FUNCTION_BLOCK FINAL FB_MiscInput EXTENDS FB_EventLogger                                            	
VAR_IN_OUT                                          	
	Control					: ST_System;            	//Machine Control Instance
END_VAR                                             	                                           	
VAR           
	_Input		AT %I*		: BOOL;						//Raw Input 1
	_Input2		AT %I*		: BOOL;						//Raw Input 2                                   	
	_ManOn					: BOOL;	     				//Manual On
	_ManOff					: BOOL;	     				//Manual Off
	_ForceOn				: BOOL;	     				//Force On
	_ForceOff				: BOOL;	     				//Force Off
	_Fault					: BOOL;	     				//Device Fault
	_SimInput				: BOOL;						//Simulates Input
	_FallingEdge			: BOOL;						//Falling Edge of Value Signal
	_RisingEdge				: BOOL;						//Raising Edge of Value Signal
	_DebounceOn_ET			: REAL;						//Debounce On Elapsed Time
	_DebounceOff_ET			: REAL;						//Debounce Off Elapsed Time
	_FaultTimer_ET			: REAL;						//Fault timer elapsed
	_EvaluationError		: BOOL;						//Evaluation Error
	_TestPulseGeneralFault	: BOOL;						//Test Pulse General Fault
	_TestPulse1Fault		: BOOL;						//Test Pulse 1 Fault
	_TestPulse2Fault		: BOOL;						//Test Pulse 2 Fault
	_Alarm					: BOOL;						//Device Alarm
	_Warning				: BOOL;						//Device Warning
	_AlarmNum				: DINT;						//Device Alarm Number
	_WarningNum				: DINT;						//Device Warning Number
	_ConfInput				: BOOL;						//Confirgured Input
	_DebounceOn_DN			: BOOL;						//Debounce On Timer is Done
	_DebounceOff_DN			: BOOL;						//Debounce Off Timer is Done
	_RiseEdge				: R_TRIG;					//Rising Edge Value Trigger
	_FallEdge				: F_TRIG;					//Falling Edge Value Trigger
	_Value		AT %Q*		: BOOL;						//Value of Input
	_R_Trig					: ARRAY[0..9] OF R_TRIG;	//Private Rising Edge Triggers
END_VAR
VAR PERSISTENT
	_Name					: STRING[15];				//Name for HMI
	_Description			: STRING[40];				//Description for HMI
	_AlarmMute				: BOOL;						//Alarm Mute
	_TypeConfig				: E_InputTypeConfig;		//Type congifuration
	_DebounceOn_PT			: REAL;						//Debounce on timer preset time
	_DebounceOff_PT			: REAL;						//Debounce off timer preset time
	_FaultTimer_PT			: REAL;						//Fault timer preset time
END_VAR

M_TypeConfig();
M_AlarmMonitor();
M_WarningMonitor();
M_UnlatchManuals();

//Debounce On Timer
IF _ConfInput = TRUE AND NOT _ForceOff AND NOT _ManOff THEN
	_DebounceOn_ET := _DebounceOn_ET + Control.SystemTime.ScanTime;
	_debounceOn_DN := _DebounceOn_ET > _DebounceOn_PT;
ELSE
	_debounceOn_DN := FALSE;
END_IF
IF _debounceOn_DN OR _ForceOn OR _ManOn THEN
	_Value := TRUE;
	_DebounceOff_ET := 0;
END_IF

//Debounce Off Timer
IF _ConfInput = FALSE AND NOT _ForceOn AND NOT _ManOn THEN
	_DebounceOff_ET := _DebounceOff_ET + Control.SystemTime.ScanTime;
	_debounceOff_DN := _DebounceOff_ET > _DebounceOff_PT;
ELSE
	_debounceOff_DN := FALSE;
END_IF
IF _debounceOff_DN OR _ForceOff OR _ManOff THEN
	_Value := FALSE;
	_DebounceOn_ET := 0;
END_IF

//Rising Edge Trigger 
_riseEdge(CLK := _Value);
_RisingEdge := _riseEdge.Q;

//Falling Edge Trigger
_fallEdge(CLK := _Value);
_FallingEdge := _fallEdge.Q;

{attribute 'monitoring' := 'variable'}
PROPERTY PUBLIC Alarm : Bool
GET
Alarm := _Alarm;
END_GET
END_PROPERTY

{attribute 'monitoring' := 'variable'}
PROPERTY PUBLIC AlarmMute : BOOL
SET
AlarmMute := _AlarmMute;
END_SET
END_PROPERTY

{attribute 'monitoring' := 'variable'}
PROPERTY PUBLIC AutoStandbyReset : Bool
GET
AutoStandbyReset := _ForceOff;
END_GET
SET
_ForceOff := AutoStandbyReset;
END_SET
END_PROPERTY

{attribute 'monitoring' := 'variable'}
PROPERTY PUBLIC DebounceOff_ET : real
GET
DebounceOff_ET := _DebounceOff_ET;
END_GET
END_PROPERTY

{attribute 'monitoring' := 'variable'}
PROPERTY PUBLIC DebounceOff_PT : real
GET
DebounceOff_PT := _DebounceOff_PT;
END_GET
SET
_DebounceOff_PT := DebounceOff_PT;
END_SET
END_PROPERTY

{attribute 'monitoring' := 'variable'}
PROPERTY PUBLIC DebounceOn_ET : real
GET
DebounceOn_ET := _DebounceOn_ET;
END_GET
END_PROPERTY

{attribute 'monitoring' := 'variable'}
PROPERTY PUBLIC DebounceOn_PT : real
GET
DebounceOn_PT := _DebounceOn_PT;
END_GET
SET
_DebounceOn_PT := DebounceOn_PT;
END_SET
END_PROPERTY

{attribute 'monitoring' := 'variable'}
PROPERTY PUBLIC Description : String[40]
GET
Description := _Description;
END_GET
SET
_Description := Description;
END_SET
END_PROPERTY

{attribute 'monitoring' := 'variable'}
PROPERTY PUBLIC EvaluationError : Bool
GET // PUBLIC
EvaluationError := _EvaluationError;
END_GET
SET
_EvaluationError := EvaluationError;
END_SET
END_PROPERTY

{attribute 'monitoring' := 'variable'}
PROPERTY PUBLIC FallingEdge : Bool
GET
FallingEdge := _FallingEdge;
END_GET
END_PROPERTY

{attribute 'monitoring' := 'variable'}
PROPERTY PUBLIC Fault : Bool
SET
_Fault := Fault;
END_SET
END_PROPERTY

{attribute 'monitoring' := 'variable'}
PROPERTY PUBLIC FaultTimer_ET : real
GET
FaultTimer_ET := _FaultTimer_ET;
END_GET
END_PROPERTY

{attribute 'monitoring' := 'variable'}
PROPERTY PUBLIC FaultTimer_PT : real
GET
FaultTimer_PT := _FaultTimer_PT;
END_GET
SET
_FaultTimer_PT := FaultTimer_PT;
END_SET
END_PROPERTY

{attribute 'monitoring' := 'variable'}
PROPERTY PUBLIC ForceOn : Bool
GET
ForceOn := _ForceOn;
END_GET
SET
_ForceOn := ForceOn;
END_SET
END_PROPERTY

{attribute 'monitoring' := 'variable'}
PROPERTY PUBLIC Input : Bool
GET
Input := _Input;
END_GET
SET // PUBLIC
_Input := Input;
END_SET
END_PROPERTY

{attribute 'monitoring' := 'variable'}
PROPERTY PUBLIC Input2 : Bool
GET
Input2 := _Input2;
END_GET
END_PROPERTY

METHOD PRIVATE M_AlarmMonitor
VAR_INPUT
END_VAR
VAR_INST
	_EvaluationError_TON		: 		TON;
END_VAR
VAR_INST // added by the converter: edge detectors and wires of the graphical bodies
    _w1, _w2, _w3, _w4, _w5 : BOOL;
    _rt1 : R_TRIG;
END_VAR
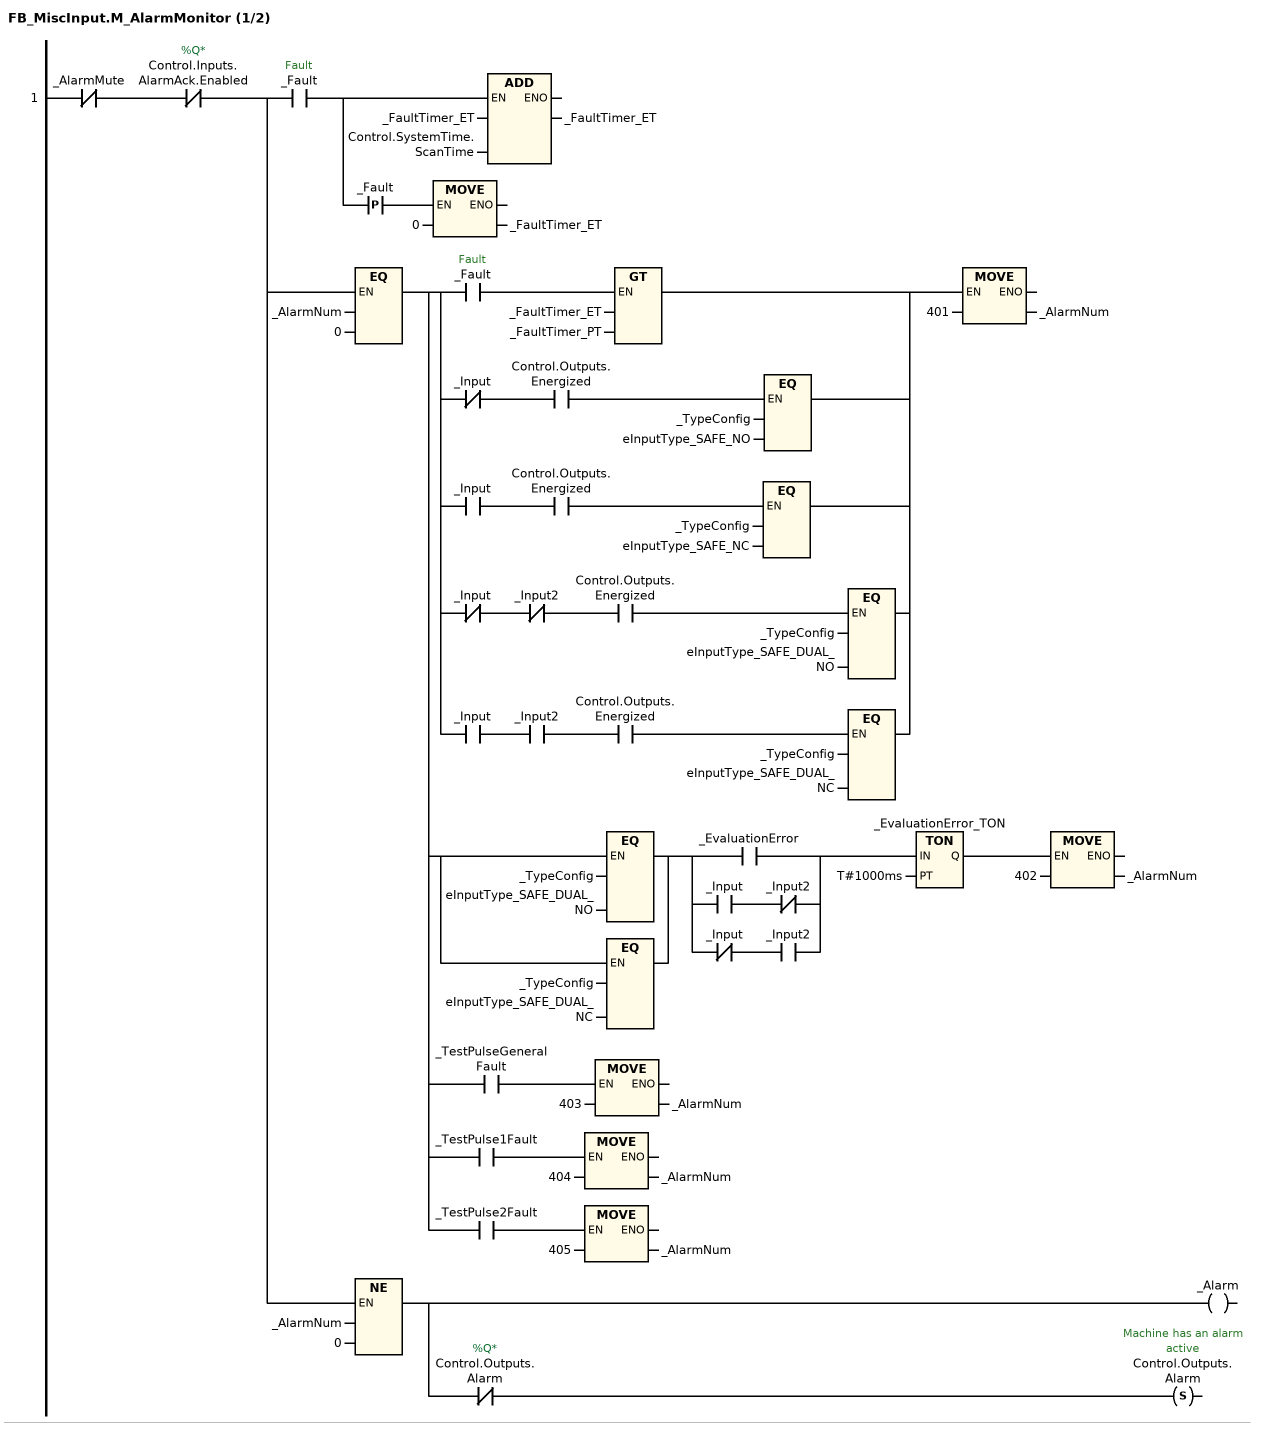
// NETWORK 1
//   Control.Inputs.AlarmAck.Enabled: AT %Q*
//   _Fault: Fault
//   _FaultTimer_ET: Fault timer elapsed
//   Control.SystemTime.ScanTime: Last scan time (Seconds)
//   _FaultTimer_PT: Fault timer preset time
//   Control.Outputs.Alarm: AT %Q* | Machine has an alarm active
_w1 := NOT _AlarmMute AND NOT Control.Inputs.AlarmAck.Enabled;
_w2 := _w1 AND _Fault;
IF _w2 THEN _FaultTimer_ET := _FaultTimer_ET + Control.SystemTime.ScanTime; END_IF
_rt1(CLK := _Fault);
IF _w2 AND _rt1.Q THEN _FaultTimer_ET := 0; END_IF
_w3 := _w1 AND _AlarmNum = 0;
IF _w3 AND _Fault AND _FaultTimer_ET > _FaultTimer_PT OR (_w3 AND NOT _Input) AND Control.Outputs.Energized AND _TypeConfig = eInputType_SAFE_NO OR (_w3 AND _Input) AND Control.Outputs.Energized AND _TypeConfig = eInputType_SAFE_NC OR (_w3 AND NOT _Input) AND NOT _Input2 AND Control.Outputs.Energized AND _TypeConfig = eInputType_SAFE_DUAL_NO OR (_w3 AND _Input) AND _Input2 AND Control.Outputs.Energized AND _TypeConfig = eInputType_SAFE_DUAL_NC THEN
    _AlarmNum := 401;
END_IF
_EvaluationError_TON(IN := (_w3 AND _TypeConfig = eInputType_SAFE_DUAL_NO OR _w3 AND _TypeConfig = eInputType_SAFE_DUAL_NC) AND (_EvaluationError OR _Input AND NOT _Input2 OR NOT _Input AND _Input2), PT := T#1000ms); // TON
IF _EvaluationError_TON.Q THEN _AlarmNum := 402; END_IF
IF _w3 AND _TestPulseGeneralFault THEN _AlarmNum := 403; END_IF
IF _w3 AND _TestPulse1Fault THEN _AlarmNum := 404; END_IF
IF _w3 AND _TestPulse2Fault THEN _AlarmNum := 405; END_IF
_w4 := _w1 AND _AlarmNum <> 0;
_Alarm := _w4;
Control.Outputs.Alarm S= _w4 AND NOT Control.Outputs.Alarm;

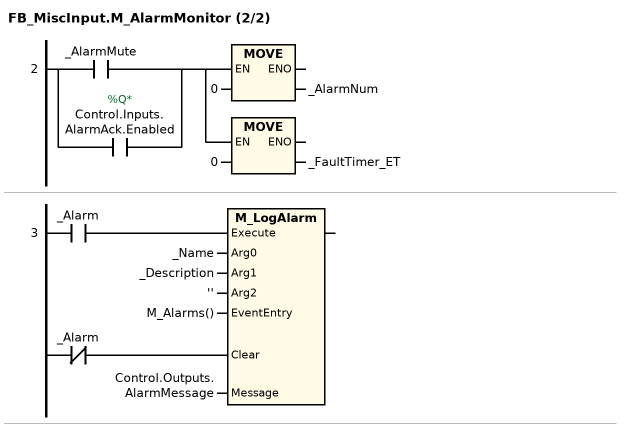
// NETWORK 2
//   Control.Inputs.AlarmAck.Enabled: AT %Q*
//   _FaultTimer_ET: Fault timer elapsed
_w5 := _AlarmMute OR Control.Inputs.AlarmAck.Enabled;
IF _w5 THEN _AlarmNum := 0; END_IF
IF _w5 THEN _FaultTimer_ET := 0; END_IF

// NETWORK 3
M_LogAlarm(Execute := _Alarm, Arg0 := _Name, Arg1 := _Description, Arg2 := '', EventEntry := M_Alarms(), Clear := NOT _Alarm, Message := Control.Outputs.AlarmMessage);
END_METHOD

METHOD PRIVATE M_Alarms : TcEventEntry
VAR_INPUT
END_VAR
CASE _AlarmNum OF
	401: M_Alarms:= TC_Events.TcMiscInput.A_401;//Alarm
	402: M_Alarms:= TC_Events.TcMiscInput.A_402;//Evaluation Error. Contact 1 or 2 failed to switch or switched too late			
	403: M_Alarms:= TC_Events.TcMiscInput.A_403;//Error in the test pulse wiring.
	404: M_Alarms:= TC_Events.TcMiscInput.A_404;//Channel 1 Input Test Pulse Error	
	405: M_Alarms:= TC_Events.TcMiscInput.A_405;//Channel 2 Input Test Pulse Error			
	406: M_Alarms:= TC_Events.TcMiscInput.A_406;//Expected to be ON Fault		
	407: M_Alarms:= TC_Events.TcMiscInput.A_407;//Expected to be OFF Fault						
ELSE
	M_Alarms:= TC_Events.TcMiscInput.A_Undefined;
END_CASE
END_METHOD

METHOD PRIVATE M_TypeConfig
VAR_INPUT
END_VAR
VAR_INST
END_VAR
CASE _TypeConfig OF
	eInputType_PLC_NO, eInputType_SAFE_NO : 
		IF _Input OR _SimInput THEN
			_ConfInput := TRUE;
		ELSE
			_ConfInput := FALSE;
		END_IF
	eInputType_PLC_NC, eInputType_SAFE_NC : 
		IF NOT _Input OR _SimInput THEN
			_ConfInput := TRUE;
		ELSE
			_ConfInput := FALSE;
		END_IF
	eInputType_SAFE_DUAL_NO : 
		IF _Input AND _Input2 THEN
			_ConfInput := TRUE;
		ELSE
			_ConfInput := FALSE;
		END_IF
	eInputType_SAFE_DUAL_NC : 
		IF NOT _Input AND NOT _Input2 THEN
			_ConfInput := TRUE;
		ELSE
			_ConfInput := FALSE;
		END_IF
	eInputType_SAFE_DUAL_NO_NC : 
		IF _Input AND NOT _Input2 THEN
			_ConfInput := TRUE;
		ELSE
			_ConfInput := FALSE;
		END_IF
END_CASE
END_METHOD

METHOD PRIVATE M_UnlatchManuals
VAR_INPUT
END_VAR
VAR_INST
END_VAR
VAR_INST // added by the converter: edge detectors and wires of the graphical bodies
    _rt1, _rt2, _rt3 : R_TRIG;
END_VAR
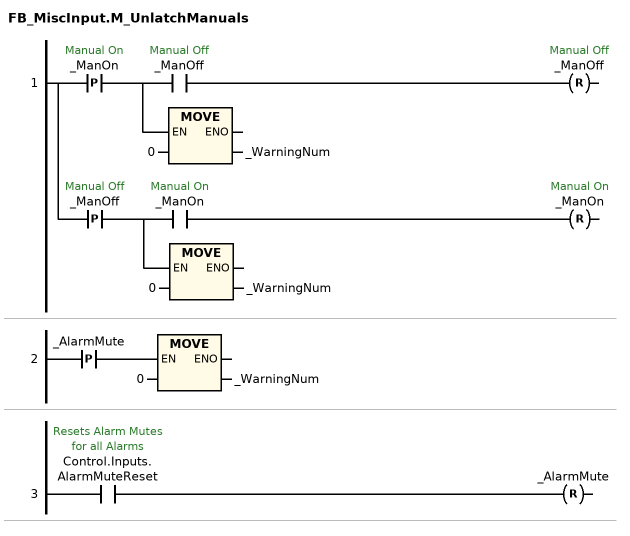
// NETWORK 1
//   _ManOn: Manual On
//   _ManOff: Manual Off
_rt1(CLK := _ManOn);
_ManOff R= _rt1.Q AND _ManOff;
IF _rt1.Q THEN _WarningNum := 0; END_IF
_rt2(CLK := _ManOff);
_ManOn R= _rt2.Q AND _ManOn;
IF _rt2.Q THEN _WarningNum := 0; END_IF

// NETWORK 2
_rt3(CLK := _AlarmMute);
IF _rt3.Q THEN _WarningNum := 0; END_IF

// NETWORK 3
//   Control.Inputs.AlarmMuteReset: Resets Alarm Mutes for all Alarms
_AlarmMute R= Control.Inputs.AlarmMuteReset;
END_METHOD

METHOD PRIVATE M_WarningMonitor
VAR_INPUT
END_VAR
VAR_INST
END_VAR
VAR_INST // added by the converter: edge detectors and wires of the graphical bodies
    _w1 : BOOL;
END_VAR
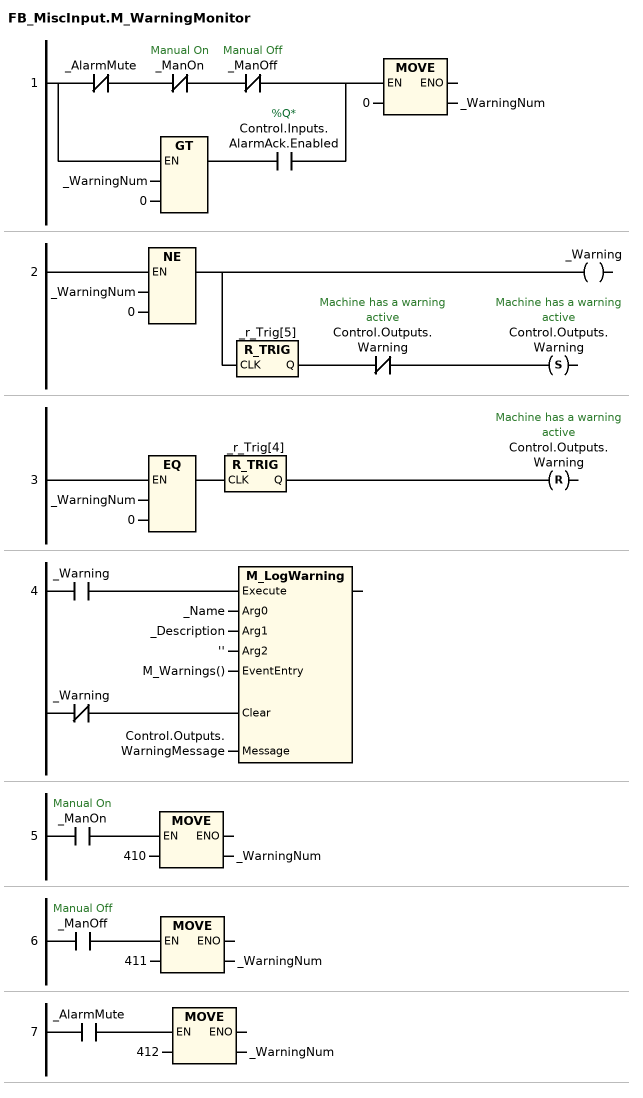
// NETWORK 1
//   _ManOn: Manual On
//   _ManOff: Manual Off
//   Control.Inputs.AlarmAck.Enabled: AT %Q*
IF NOT _AlarmMute AND NOT _ManOn AND NOT _ManOff OR _WarningNum > 0 AND Control.Inputs.AlarmAck.Enabled THEN
    _WarningNum := 0;
END_IF

// NETWORK 2
//   Control.Outputs.Warning: Machine has a warning active
_w1 := _WarningNum <> 0;
_Warning := _w1;
_r_Trig[5](CLK := _w1); // R_TRIG
Control.Outputs.Warning S= _r_Trig[5].Q AND NOT Control.Outputs.Warning;

// NETWORK 3
//   Control.Outputs.Warning: Machine has a warning active
_r_Trig[4](CLK := _WarningNum = 0); // R_TRIG
Control.Outputs.Warning R= _r_Trig[4].Q;

// NETWORK 4
M_LogWarning(Execute := _Warning, Arg0 := _Name, Arg1 := _Description, Arg2 := '', EventEntry := M_Warnings(), Clear := NOT _Warning, Message := Control.Outputs.WarningMessage);

// NETWORK 5
//   _ManOn: Manual On
IF _ManOn THEN _WarningNum := 410; END_IF

// NETWORK 6
//   _ManOff: Manual Off
IF _ManOff THEN _WarningNum := 411; END_IF

// NETWORK 7
IF _AlarmMute THEN _WarningNum := 412; END_IF
END_METHOD

METHOD PRIVATE M_Warnings : TcEventEntry
VAR_INPUT
END_VAR
CASE _WarningNum OF
	410: M_Warnings:= TC_Events.TcMiscInput.W_410;//Manual ON Enabled	
	411: M_Warnings:= TC_Events.TcMiscInput.W_411;//Manual OFF Enabled			
	412: M_Warnings:= TC_Events.TcMiscInput.W_412;//Alarm Mute Active						
ELSE
	M_Warnings:=  TC_Events.TcMiscInput.W_Undefined;
END_CASE
END_METHOD

{attribute 'monitoring' := 'variable'}
PROPERTY PUBLIC ManOff : Bool
GET
ManOff := _ManOff;
END_GET
SET
_ManOff := ManOff;
END_SET
END_PROPERTY

{attribute 'monitoring' := 'variable'}
PROPERTY PUBLIC ManOn : Bool
GET
ManOn := _ManOn;
END_GET
SET
_ManOn := ManOn;
END_SET
END_PROPERTY

{attribute 'monitoring' := 'variable'}
PROPERTY PUBLIC Name : String[15]
GET
Name := _Name;
END_GET
SET
_Name := Name;
END_SET
END_PROPERTY

{attribute 'monitoring' := 'variable'}
PROPERTY PUBLIC RisingEdge : Bool
GET
RisingEdge := _RisingEdge;
END_GET
END_PROPERTY

{attribute 'monitoring' := 'variable'}
PROPERTY PUBLIC SimInput : Bool
SET
_SimInput := SimInput;
END_SET
END_PROPERTY

{attribute 'monitoring' := 'variable'}
PROPERTY PUBLIC TestPulse1Fault : Bool
GET
TestPulse1Fault := _TestPulse1Fault;
END_GET
SET
_TestPulse1Fault := TestPulse1Fault;
END_SET
END_PROPERTY

{attribute 'monitoring' := 'variable'}
PROPERTY PUBLIC TestPulse2Fault : Bool
GET
TestPulse2Fault := _TestPulse2Fault;
END_GET
SET
_TestPulse2Fault := TestPulse2Fault;
END_SET
END_PROPERTY

{attribute 'monitoring' := 'variable'}
PROPERTY PUBLIC TestPulseGeneralFault : Bool
GET
TestPulseGeneralFault := _TestPulseGeneralFault;
END_GET
SET
_TestPulseGeneralFault := TestPulseGeneralFault;
END_SET
END_PROPERTY

{attribute 'monitoring' := 'variable'}
PROPERTY PUBLIC Value : Bool
GET
Value := _Value;
END_GET
SET
_Value := Value;
END_SET
END_PROPERTY

{attribute 'monitoring' := 'variable'}
PROPERTY PUBLIC Warning : Bool
GET
Warning := _Warning;
END_GET
END_PROPERTY

END_FUNCTION_BLOCK

(* stored: Version 1.1.0.1, ProductVersion 3.1.4024.3
   POU FB_MiscInput: Id {c0d88bc5-b182-49df-b578-ed0f16238807}, SpecialFunc None
   Property Alarm: Id {3658f6dc-6e01-4ab1-aa7a-12bbd299ad4b}
   Get Get: Id {6c509c0c-7480-4274-ae68-68e3a9df5369}
   Property AlarmMute: Id {ffa553a3-2559-4579-a69b-9f764a8d08ab}
   Set Set: Id {cf89d9e7-8292-4528-a66f-29cd89792830}
   Property AutoStandbyReset: Id {18cb0727-a662-4c09-8dbc-84357f54838e}
   Get Get: Id {b0a025ea-2b9e-400d-8a61-1d76b1ed73bf}
   Set Set: Id {b2ad94f4-5c45-4b2e-82a5-1581ac1c5dc8}
   Property DebounceOff_ET: Id {74509f44-dd39-4467-8d20-707144248c24}
   Get Get: Id {54d68720-48e0-4727-905c-29fbd4979d9a}
   Property DebounceOff_PT: Id {59f53b24-f1c7-4249-805f-05c62da47c84}
   Get Get: Id {8891ec69-8d1f-4c4a-b114-deeb08ce2fb7}
   Set Set: Id {ed01c235-50fd-48e7-b591-2a2a9a9e33ce}
   Property DebounceOn_ET: Id {41af56ee-a2d6-477e-b0cf-98933ddbaa42}
   Get Get: Id {cbd68782-1d64-467e-aabe-68254bed39b3}
   Property DebounceOn_PT: Id {251423d0-2084-4b2d-afa5-afd07bfcc653}
   Get Get: Id {a8f1dbac-0971-46e9-9af2-c1757fd9c4f5}
   Set Set: Id {d501fff4-40d2-4cda-bdf5-80cb053ebb49}
   Property Description: Id {0a20c4d0-0852-4169-8173-d3c2bd3caa54}
   Get Get: Id {124a4c05-8915-484c-b001-008a20669f39}
   Set Set: Id {f84e5111-a402-48fd-a46f-f4a9cee7eb8c}
   Property EvaluationError: Id {f8c56a30-f5c7-41f6-aee7-0206f6f8cd4e}
   Get Get: Id {38e8d71a-2fe3-43ac-aea2-c10b7579b2e9}
   Set Set: Id {ff11a864-f0e3-4f8f-acd7-475b40d97727}
   Property FallingEdge: Id {1dd8b317-91a8-4de8-b759-d4e8f3ca831a}
   Get Get: Id {e6170223-0c69-4d8c-8877-6cf3fd201983}
   Property Fault: Id {125dc8d1-6763-4ef4-93a0-c88b685b439a}
   Set Set: Id {ae2cc827-cc43-4139-bb37-9ded44db5652}
   Property FaultTimer_ET: Id {0fba5d22-2aeb-4884-b5c9-eb62bc396633}
   Get Get: Id {1111c4e2-66c0-4d9f-9925-39545e35947a}
   Property FaultTimer_PT: Id {d2d56292-bc61-416b-8e16-e19ad9993c6e}
   Get Get: Id {34faa55f-4d25-41b6-883c-99de9ba5fb41}
   Set Set: Id {daca9458-4a85-4640-982b-cf6448678cba}
   Property ForceOn: Id {0377b997-3862-47a0-95f4-b96c26817522}
   Get Get: Id {06c3b5dc-e414-4a3a-a58e-0c0a4672b0ad}
   Set Set: Id {a0ce7201-4ff4-408a-a056-42104c48bc78}
   Property Input: Id {488231ea-c389-4dd6-8b10-b85cda51d1dc}
   Get Get: Id {55032826-2e2a-4ab2-919c-0cd7931ef0fa}
   Set Set: Id {00a98704-90c3-4ab5-9755-e1394caca87d}
   Property Input2: Id {a441fdbc-27f5-4bd6-a1bf-204e52cb7712}
   Get Get: Id {a0d87452-58a1-4b2b-8b9c-f140e2cdba22}
   Method M_AlarmMonitor: Id {7ca0b0a4-1432-430e-b009-7d687ad3806f}
   Method M_Alarms: Id {c867b0f2-aa9f-49f4-96fa-dbbc2082d479}
   Method M_TypeConfig: Id {4a7e9782-dd7a-4141-992d-c79556985019}
   Method M_UnlatchManuals: Id {2bd763b3-55d1-4150-b0ec-e296a1f80358}
   Method M_WarningMonitor: Id {583cee2f-f972-4331-a8ee-8fba29d76a89}
   Method M_Warnings: Id {f0c100d2-055b-4c71-a5ca-5744cfb67d26}
   Property ManOff: Id {18c427a3-b5f4-49d8-8024-d24d3e51a681}
   Get Get: Id {2c36e6a8-0f41-487f-b4d1-51c40bc21ef1}
   Set Set: Id {2573b357-9d4f-41f5-8737-2fbb1dd13605}
   Property ManOn: Id {0e133ec4-1599-4ebb-b406-35e05fb2c0bb}
   Get Get: Id {7df83b3c-429d-496b-a33a-656de7942966}
   Set Set: Id {eba54b43-038e-46b3-bde0-df3e437c05f8}
   Property Name: Id {23ff72d4-11f9-447d-b9b1-0b8adf36daaa}
   Get Get: Id {17028a0b-910a-49b3-a4c1-72fd230b2f75}
   Set Set: Id {84d80d55-f619-4c80-ac5a-5c0f5305badd}
   Property RisingEdge: Id {97e0f4e1-a76f-4f1e-a85d-3e5217da4311}
   Get Get: Id {a415b987-98ac-4008-94ee-3e79e7da5f22}
   Property SimInput: Id {9ebabc78-61d5-4206-8c01-1ed75c8ddc37}
   Set Set: Id {79f2d6dc-d603-46a9-9b25-dff54633376d}
   Property TestPulse1Fault: Id {1257884c-241b-4688-b191-2f7851d64552}
   Get Get: Id {5aa6dd55-2a4a-4b70-9a90-6cf6932f1510}
   Set Set: Id {5ad4321c-d951-4bce-8769-09d5240708f9}
   Property TestPulse2Fault: Id {860feba9-c546-4aa1-acf7-8b8ce19afe6d}
   Get Get: Id {62c0668d-0b57-4ce2-92c0-46a414a5dfd9}
   Set Set: Id {9c71f304-5028-47ce-86e8-89e024f8b88e}
   Property TestPulseGeneralFault: Id {8056dc54-5025-4c99-b4e6-379fafd46543}
   Get Get: Id {a586ab93-a57d-4471-b769-a4a332ae4ae1}
   Set Set: Id {882c23ef-103c-415f-b28b-14ab4e646206}
   Property Value: Id {2da36000-5614-4d3f-a9ac-ba1138f1d2a4}
   Get Get: Id {760034b7-0e88-4199-9ef2-a7f37e0f5cb6}
   Set Set: Id {1bf0230b-062e-428c-a564-40a334c97b34}
   Property Warning: Id {7d81033a-c0dc-4f30-bb79-273c68c87206}
   Get Get: Id {c267b1fa-9044-4d7e-8595-4b5d5f82fd7c} *)
